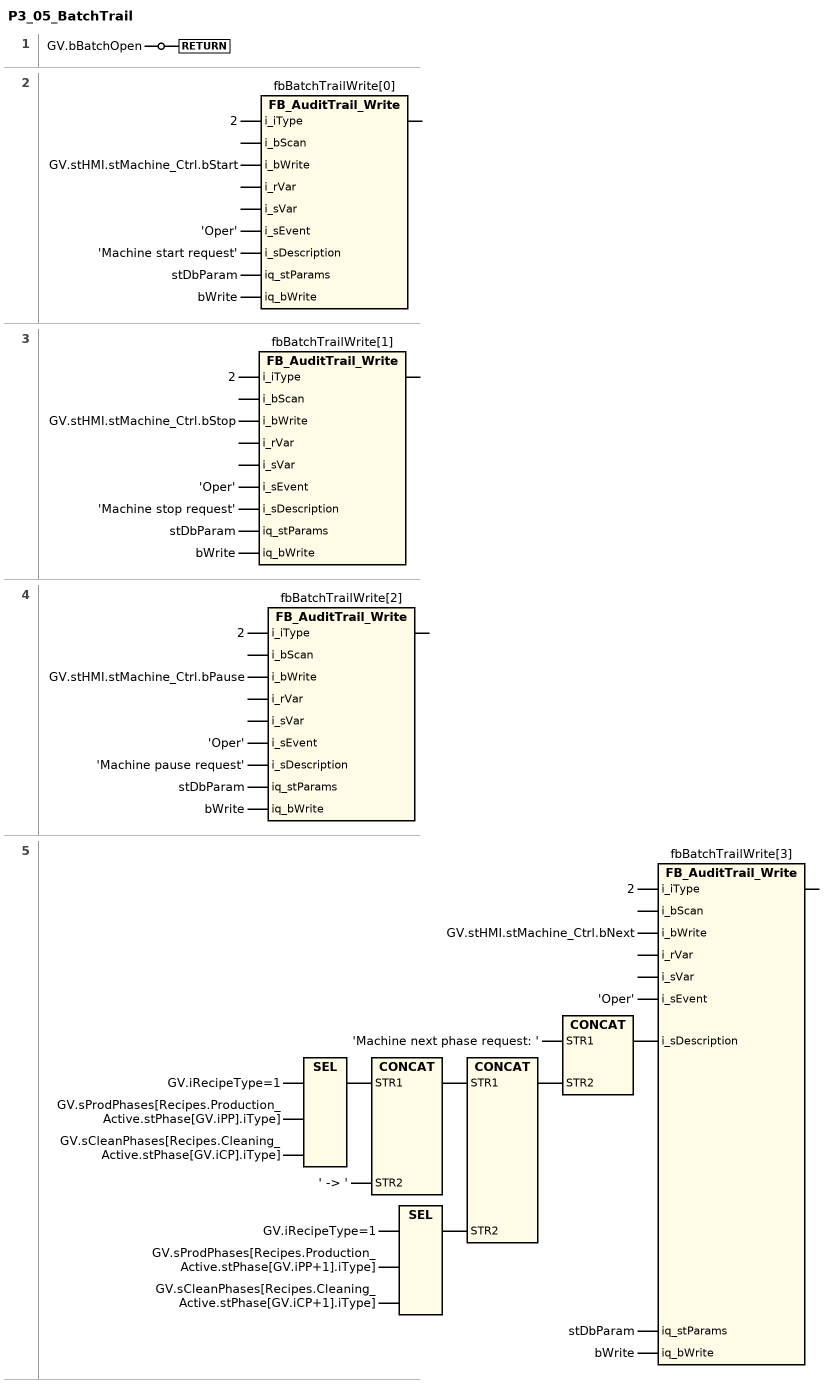
// NETWORK 1
IF NOT GV.bBatchOpen THEN RETURN; END_IF

// NETWORK 2
fbBatchTrailWrite[0](
    i_iType := 2,
    i_bWrite := GV.stHMI.stMachine_Ctrl.bStart,
    i_sEvent := 'Oper',
    i_sDescription := 'Machine start request',
    iq_stParams := stDbParam,
    iq_bWrite := bWrite); // FB_AuditTrail_Write

// NETWORK 3
fbBatchTrailWrite[1](
    i_iType := 2,
    i_bWrite := GV.stHMI.stMachine_Ctrl.bStop,
    i_sEvent := 'Oper',
    i_sDescription := 'Machine stop request',
    iq_stParams := stDbParam,
    iq_bWrite := bWrite); // FB_AuditTrail_Write

// NETWORK 4
fbBatchTrailWrite[2](
    i_iType := 2,
    i_bWrite := GV.stHMI.stMachine_Ctrl.bPause,
    i_sEvent := 'Oper',
    i_sDescription := 'Machine pause request',
    iq_stParams := stDbParam,
    iq_bWrite := bWrite); // FB_AuditTrail_Write

// NETWORK 5
fbBatchTrailWrite[3](
    i_iType := 2,
    i_bWrite := GV.stHMI.stMachine_Ctrl.bNext,
    i_sEvent := 'Oper',
    i_sDescription := CONCAT(STR1 := 'Machine next phase request: ', STR2 := CONCAT(STR1 := CONCAT(STR1 := SEL(GV.iRecipeType=1, GV.sProdPhases[Recipes.Production_Active.stPhase[GV.iPP].iType], GV.sCleanPhases[Recipes.Cleaning_Active.stPhase[GV.iCP].iType]), STR2 := ' -> '), STR2 := SEL(GV.iRecipeType=1, GV.sProdPhases[Recipes.Production_Active.stPhase[GV.iPP+1].iType], GV.sCleanPhases[Recipes.Cleaning_Active.stPhase[GV.iCP+1].iType]))),
    iq_stParams := stDbParam,
    iq_bWrite := bWrite); // FB_AuditTrail_Write

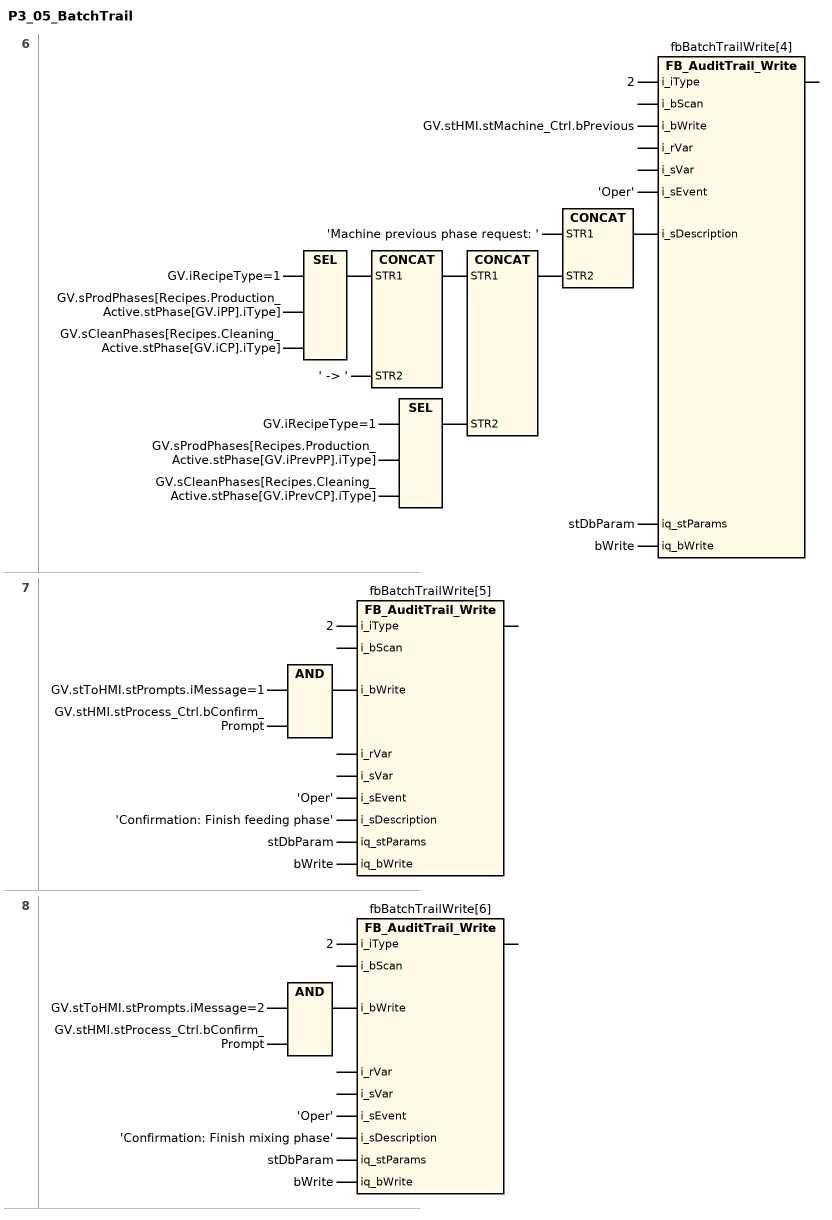
// NETWORK 6
fbBatchTrailWrite[4](
    i_iType := 2,
    i_bWrite := GV.stHMI.stMachine_Ctrl.bPrevious,
    i_sEvent := 'Oper',
    i_sDescription := CONCAT(STR1 := 'Machine previous phase request: ', STR2 := CONCAT(STR1 := CONCAT(STR1 := SEL(GV.iRecipeType=1, GV.sProdPhases[Recipes.Production_Active.stPhase[GV.iPP].iType], GV.sCleanPhases[Recipes.Cleaning_Active.stPhase[GV.iCP].iType]), STR2 := ' -> '), STR2 := SEL(GV.iRecipeType=1, GV.sProdPhases[Recipes.Production_Active.stPhase[GV.iPrevPP].iType], GV.sCleanPhases[Recipes.Cleaning_Active.stPhase[GV.iPrevCP].iType]))),
    iq_stParams := stDbParam,
    iq_bWrite := bWrite); // FB_AuditTrail_Write

// NETWORK 7
fbBatchTrailWrite[5](
    i_iType := 2,
    i_bWrite := (GV.stToHMI.stPrompts.iMessage=1) AND GV.stHMI.stProcess_Ctrl.bConfirm_Prompt,
    i_sEvent := 'Oper',
    i_sDescription := 'Confirmation: Finish feeding phase',
    iq_stParams := stDbParam,
    iq_bWrite := bWrite); // FB_AuditTrail_Write

// NETWORK 8
fbBatchTrailWrite[6](
    i_iType := 2,
    i_bWrite := (GV.stToHMI.stPrompts.iMessage=2) AND GV.stHMI.stProcess_Ctrl.bConfirm_Prompt,
    i_sEvent := 'Oper',
    i_sDescription := 'Confirmation: Finish mixing phase',
    iq_stParams := stDbParam,
    iq_bWrite := bWrite); // FB_AuditTrail_Write

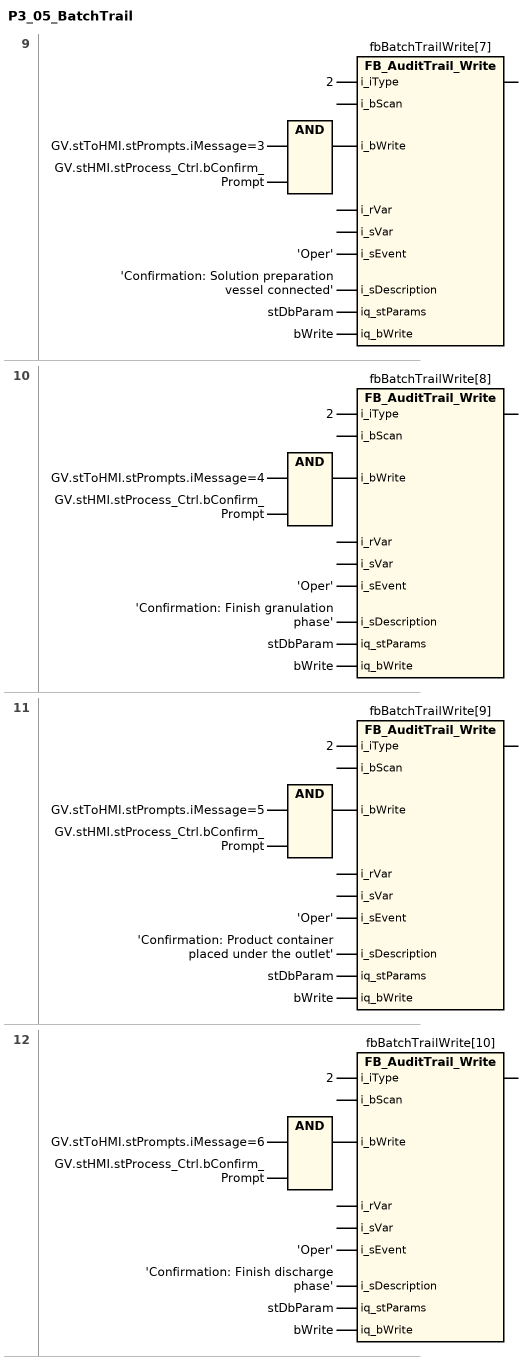
// NETWORK 9
fbBatchTrailWrite[7](
    i_iType := 2,
    i_bWrite := (GV.stToHMI.stPrompts.iMessage=3) AND GV.stHMI.stProcess_Ctrl.bConfirm_Prompt,
    i_sEvent := 'Oper',
    i_sDescription := 'Confirmation: Solution preparation vessel connected',
    iq_stParams := stDbParam,
    iq_bWrite := bWrite); // FB_AuditTrail_Write

// NETWORK 10
fbBatchTrailWrite[8](
    i_iType := 2,
    i_bWrite := (GV.stToHMI.stPrompts.iMessage=4) AND GV.stHMI.stProcess_Ctrl.bConfirm_Prompt,
    i_sEvent := 'Oper',
    i_sDescription := 'Confirmation: Finish granulation phase',
    iq_stParams := stDbParam,
    iq_bWrite := bWrite); // FB_AuditTrail_Write

// NETWORK 11
fbBatchTrailWrite[9](
    i_iType := 2,
    i_bWrite := (GV.stToHMI.stPrompts.iMessage=5) AND GV.stHMI.stProcess_Ctrl.bConfirm_Prompt,
    i_sEvent := 'Oper',
    i_sDescription := 'Confirmation: Product container placed under the outlet',
    iq_stParams := stDbParam,
    iq_bWrite := bWrite); // FB_AuditTrail_Write

// NETWORK 12
fbBatchTrailWrite[10](
    i_iType := 2,
    i_bWrite := (GV.stToHMI.stPrompts.iMessage=6) AND GV.stHMI.stProcess_Ctrl.bConfirm_Prompt,
    i_sEvent := 'Oper',
    i_sDescription := 'Confirmation: Finish discharge phase',
    iq_stParams := stDbParam,
    iq_bWrite := bWrite); // FB_AuditTrail_Write

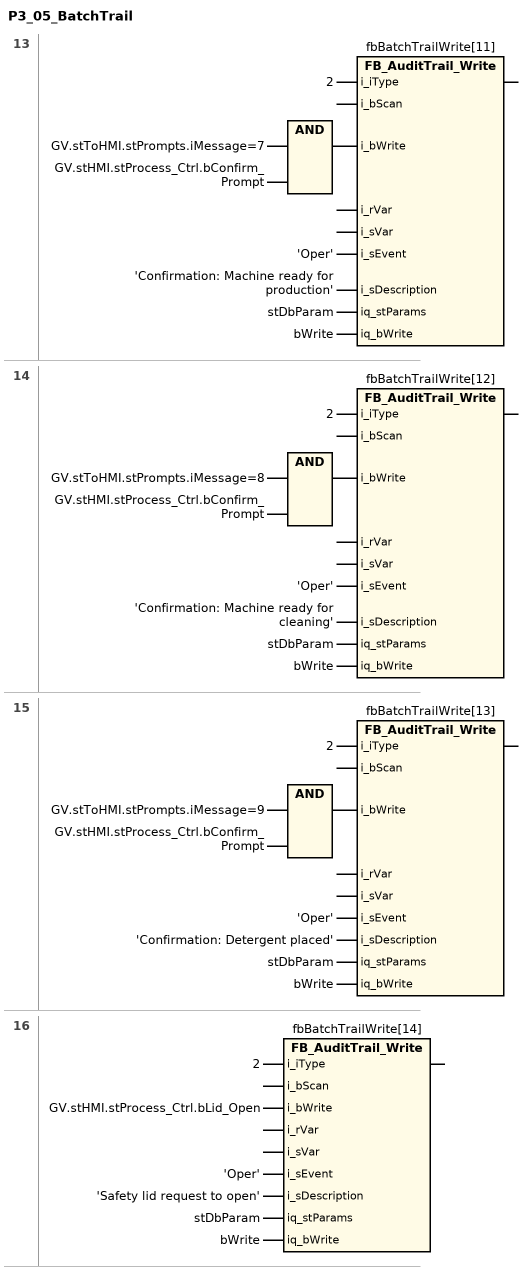
// NETWORK 13
fbBatchTrailWrite[11](
    i_iType := 2,
    i_bWrite := (GV.stToHMI.stPrompts.iMessage=7) AND GV.stHMI.stProcess_Ctrl.bConfirm_Prompt,
    i_sEvent := 'Oper',
    i_sDescription := 'Confirmation: Machine ready for production',
    iq_stParams := stDbParam,
    iq_bWrite := bWrite); // FB_AuditTrail_Write

// NETWORK 14
fbBatchTrailWrite[12](
    i_iType := 2,
    i_bWrite := (GV.stToHMI.stPrompts.iMessage=8) AND GV.stHMI.stProcess_Ctrl.bConfirm_Prompt,
    i_sEvent := 'Oper',
    i_sDescription := 'Confirmation: Machine ready for cleaning',
    iq_stParams := stDbParam,
    iq_bWrite := bWrite); // FB_AuditTrail_Write

// NETWORK 15
fbBatchTrailWrite[13](
    i_iType := 2,
    i_bWrite := (GV.stToHMI.stPrompts.iMessage=9) AND GV.stHMI.stProcess_Ctrl.bConfirm_Prompt,
    i_sEvent := 'Oper',
    i_sDescription := 'Confirmation: Detergent placed',
    iq_stParams := stDbParam,
    iq_bWrite := bWrite); // FB_AuditTrail_Write

// NETWORK 16
fbBatchTrailWrite[14](
    i_iType := 2,
    i_bWrite := GV.stHMI.stProcess_Ctrl.bLid_Open,
    i_sEvent := 'Oper',
    i_sDescription := 'Safety lid request to open',
    iq_stParams := stDbParam,
    iq_bWrite := bWrite); // FB_AuditTrail_Write

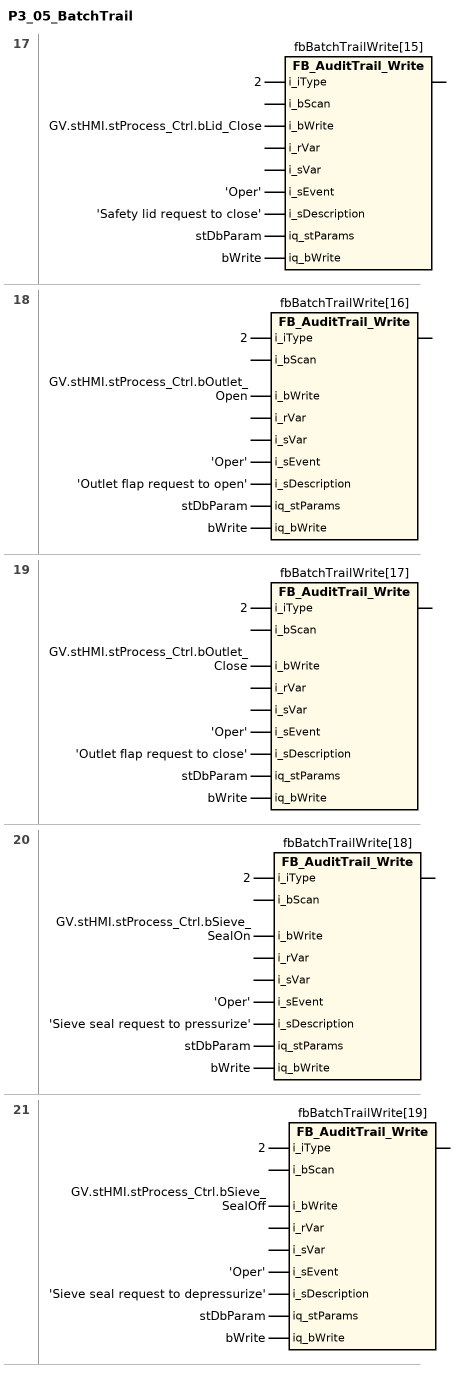
// NETWORK 17
fbBatchTrailWrite[15](
    i_iType := 2,
    i_bWrite := GV.stHMI.stProcess_Ctrl.bLid_Close,
    i_sEvent := 'Oper',
    i_sDescription := 'Safety lid request to close',
    iq_stParams := stDbParam,
    iq_bWrite := bWrite); // FB_AuditTrail_Write

// NETWORK 18
fbBatchTrailWrite[16](
    i_iType := 2,
    i_bWrite := GV.stHMI.stProcess_Ctrl.bOutlet_Open,
    i_sEvent := 'Oper',
    i_sDescription := 'Outlet flap request to open',
    iq_stParams := stDbParam,
    iq_bWrite := bWrite); // FB_AuditTrail_Write

// NETWORK 19
fbBatchTrailWrite[17](
    i_iType := 2,
    i_bWrite := GV.stHMI.stProcess_Ctrl.bOutlet_Close,
    i_sEvent := 'Oper',
    i_sDescription := 'Outlet flap request to close',
    iq_stParams := stDbParam,
    iq_bWrite := bWrite); // FB_AuditTrail_Write

// NETWORK 20
fbBatchTrailWrite[18](
    i_iType := 2,
    i_bWrite := GV.stHMI.stProcess_Ctrl.bSieve_SealOn,
    i_sEvent := 'Oper',
    i_sDescription := 'Sieve seal request to pressurize',
    iq_stParams := stDbParam,
    iq_bWrite := bWrite); // FB_AuditTrail_Write

// NETWORK 21
fbBatchTrailWrite[19](
    i_iType := 2,
    i_bWrite := GV.stHMI.stProcess_Ctrl.bSieve_SealOff,
    i_sEvent := 'Oper',
    i_sDescription := 'Sieve seal request to depressurize',
    iq_stParams := stDbParam,
    iq_bWrite := bWrite); // FB_AuditTrail_Write

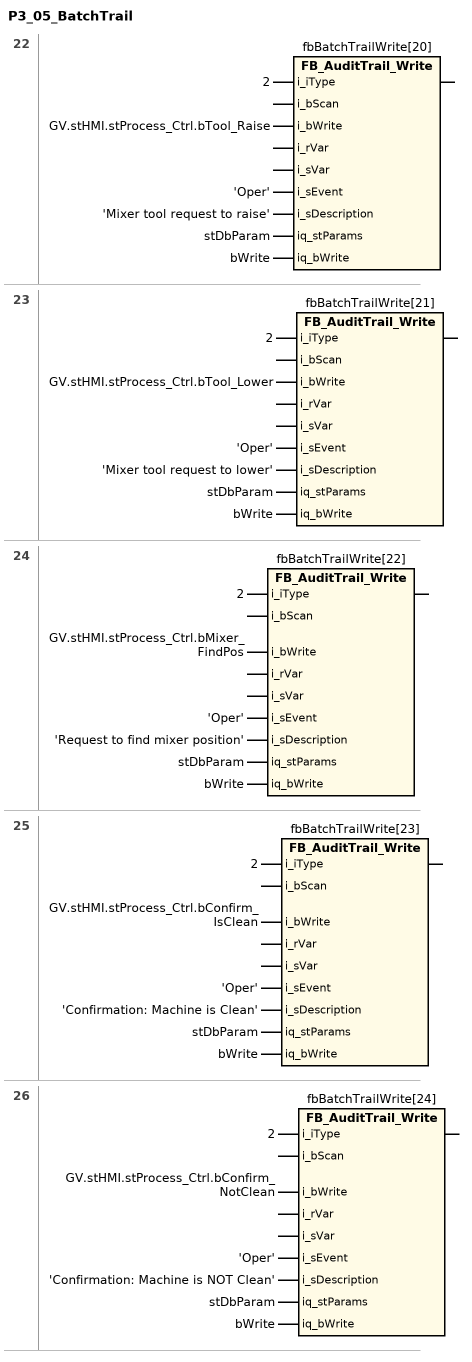
// NETWORK 22
fbBatchTrailWrite[20](
    i_iType := 2,
    i_bWrite := GV.stHMI.stProcess_Ctrl.bTool_Raise,
    i_sEvent := 'Oper',
    i_sDescription := 'Mixer tool request to raise',
    iq_stParams := stDbParam,
    iq_bWrite := bWrite); // FB_AuditTrail_Write

// NETWORK 23
fbBatchTrailWrite[21](
    i_iType := 2,
    i_bWrite := GV.stHMI.stProcess_Ctrl.bTool_Lower,
    i_sEvent := 'Oper',
    i_sDescription := 'Mixer tool request to lower',
    iq_stParams := stDbParam,
    iq_bWrite := bWrite); // FB_AuditTrail_Write

// NETWORK 24
fbBatchTrailWrite[22](
    i_iType := 2,
    i_bWrite := GV.stHMI.stProcess_Ctrl.bMixer_FindPos,
    i_sEvent := 'Oper',
    i_sDescription := 'Request to find mixer position',
    iq_stParams := stDbParam,
    iq_bWrite := bWrite); // FB_AuditTrail_Write

// NETWORK 25
fbBatchTrailWrite[23](
    i_iType := 2,
    i_bWrite := GV.stHMI.stProcess_Ctrl.bConfirm_IsClean,
    i_sEvent := 'Oper',
    i_sDescription := 'Confirmation: Machine is Clean',
    iq_stParams := stDbParam,
    iq_bWrite := bWrite); // FB_AuditTrail_Write

// NETWORK 26
fbBatchTrailWrite[24](
    i_iType := 2,
    i_bWrite := GV.stHMI.stProcess_Ctrl.bConfirm_NotClean,
    i_sEvent := 'Oper',
    i_sDescription := 'Confirmation: Machine is NOT Clean',
    iq_stParams := stDbParam,
    iq_bWrite := bWrite); // FB_AuditTrail_Write

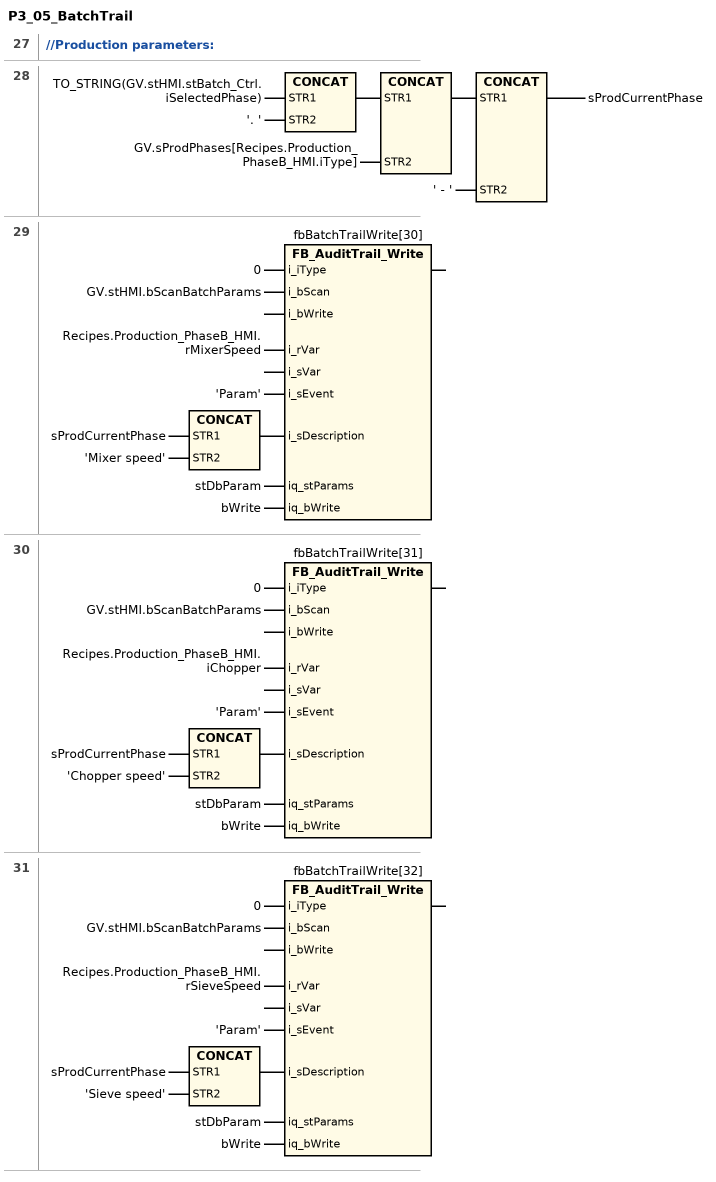
// NETWORK 27
// label: //Production parameters

// NETWORK 28
sProdCurrentPhase := CONCAT(STR1 := CONCAT(STR1 := CONCAT(STR1 := TO_STRING(GV.stHMI.stBatch_Ctrl.iSelectedPhase), STR2 := '. '), STR2 := GV.sProdPhases[Recipes.Production_PhaseB_HMI.iType]), STR2 := ' - ');

// NETWORK 29
fbBatchTrailWrite[30](
    i_iType := 0,
    i_bScan := GV.stHMI.bScanBatchParams,
    i_rVar := Recipes.Production_PhaseB_HMI.rMixerSpeed,
    i_sEvent := 'Param',
    i_sDescription := CONCAT(STR1 := sProdCurrentPhase, STR2 := 'Mixer speed'),
    iq_stParams := stDbParam,
    iq_bWrite := bWrite); // FB_AuditTrail_Write

// NETWORK 30
fbBatchTrailWrite[31](
    i_iType := 0,
    i_bScan := GV.stHMI.bScanBatchParams,
    i_rVar := Recipes.Production_PhaseB_HMI.iChopper,
    i_sEvent := 'Param',
    i_sDescription := CONCAT(STR1 := sProdCurrentPhase, STR2 := 'Chopper speed'),
    iq_stParams := stDbParam,
    iq_bWrite := bWrite); // FB_AuditTrail_Write

// NETWORK 31
fbBatchTrailWrite[32](
    i_iType := 0,
    i_bScan := GV.stHMI.bScanBatchParams,
    i_rVar := Recipes.Production_PhaseB_HMI.rSieveSpeed,
    i_sEvent := 'Param',
    i_sDescription := CONCAT(STR1 := sProdCurrentPhase, STR2 := 'Sieve speed'),
    iq_stParams := stDbParam,
    iq_bWrite := bWrite); // FB_AuditTrail_Write

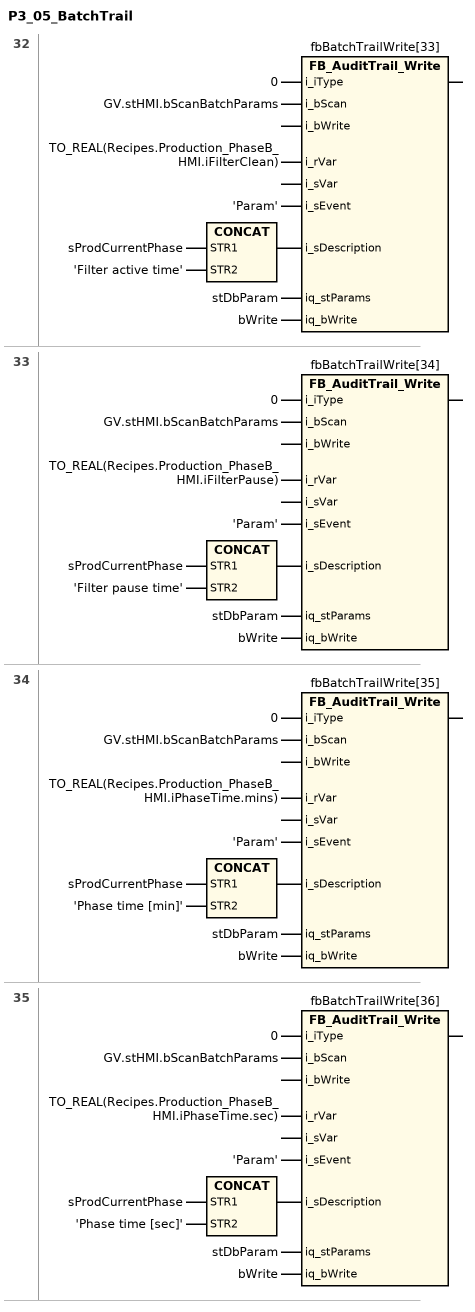
// NETWORK 32
fbBatchTrailWrite[33](
    i_iType := 0,
    i_bScan := GV.stHMI.bScanBatchParams,
    i_rVar := TO_REAL(Recipes.Production_PhaseB_HMI.iFilterClean),
    i_sEvent := 'Param',
    i_sDescription := CONCAT(STR1 := sProdCurrentPhase, STR2 := 'Filter active time'),
    iq_stParams := stDbParam,
    iq_bWrite := bWrite); // FB_AuditTrail_Write

// NETWORK 33
fbBatchTrailWrite[34](
    i_iType := 0,
    i_bScan := GV.stHMI.bScanBatchParams,
    i_rVar := TO_REAL(Recipes.Production_PhaseB_HMI.iFilterPause),
    i_sEvent := 'Param',
    i_sDescription := CONCAT(STR1 := sProdCurrentPhase, STR2 := 'Filter pause time'),
    iq_stParams := stDbParam,
    iq_bWrite := bWrite); // FB_AuditTrail_Write

// NETWORK 34
fbBatchTrailWrite[35](
    i_iType := 0,
    i_bScan := GV.stHMI.bScanBatchParams,
    i_rVar := TO_REAL(Recipes.Production_PhaseB_HMI.iPhaseTime.mins),
    i_sEvent := 'Param',
    i_sDescription := CONCAT(STR1 := sProdCurrentPhase, STR2 := 'Phase time [min]'),
    iq_stParams := stDbParam,
    iq_bWrite := bWrite); // FB_AuditTrail_Write

// NETWORK 35
fbBatchTrailWrite[36](
    i_iType := 0,
    i_bScan := GV.stHMI.bScanBatchParams,
    i_rVar := TO_REAL(Recipes.Production_PhaseB_HMI.iPhaseTime.sec),
    i_sEvent := 'Param',
    i_sDescription := CONCAT(STR1 := sProdCurrentPhase, STR2 := 'Phase time [sec]'),
    iq_stParams := stDbParam,
    iq_bWrite := bWrite); // FB_AuditTrail_Write

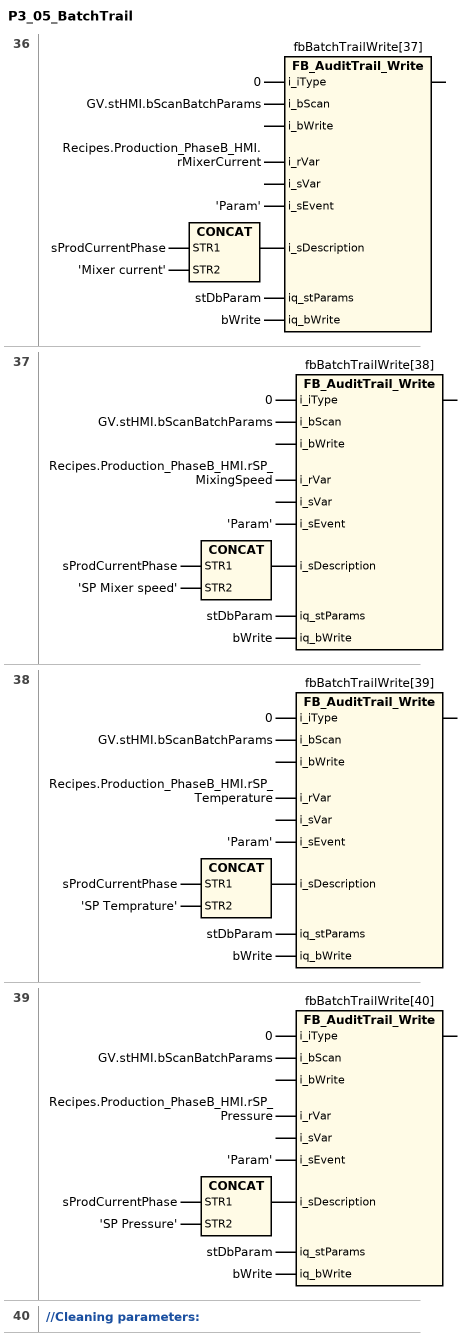
// NETWORK 36
fbBatchTrailWrite[37](
    i_iType := 0,
    i_bScan := GV.stHMI.bScanBatchParams,
    i_rVar := Recipes.Production_PhaseB_HMI.rMixerCurrent,
    i_sEvent := 'Param',
    i_sDescription := CONCAT(STR1 := sProdCurrentPhase, STR2 := 'Mixer current'),
    iq_stParams := stDbParam,
    iq_bWrite := bWrite); // FB_AuditTrail_Write

// NETWORK 37
fbBatchTrailWrite[38](
    i_iType := 0,
    i_bScan := GV.stHMI.bScanBatchParams,
    i_rVar := Recipes.Production_PhaseB_HMI.rSP_MixingSpeed,
    i_sEvent := 'Param',
    i_sDescription := CONCAT(STR1 := sProdCurrentPhase, STR2 := 'SP Mixer speed'),
    iq_stParams := stDbParam,
    iq_bWrite := bWrite); // FB_AuditTrail_Write

// NETWORK 38
fbBatchTrailWrite[39](
    i_iType := 0,
    i_bScan := GV.stHMI.bScanBatchParams,
    i_rVar := Recipes.Production_PhaseB_HMI.rSP_Temperature,
    i_sEvent := 'Param',
    i_sDescription := CONCAT(STR1 := sProdCurrentPhase, STR2 := 'SP Temprature'),
    iq_stParams := stDbParam,
    iq_bWrite := bWrite); // FB_AuditTrail_Write

// NETWORK 39
fbBatchTrailWrite[40](
    i_iType := 0,
    i_bScan := GV.stHMI.bScanBatchParams,
    i_rVar := Recipes.Production_PhaseB_HMI.rSP_Pressure,
    i_sEvent := 'Param',
    i_sDescription := CONCAT(STR1 := sProdCurrentPhase, STR2 := 'SP Pressure'),
    iq_stParams := stDbParam,
    iq_bWrite := bWrite); // FB_AuditTrail_Write

// NETWORK 40
// label: //Cleaning parameters

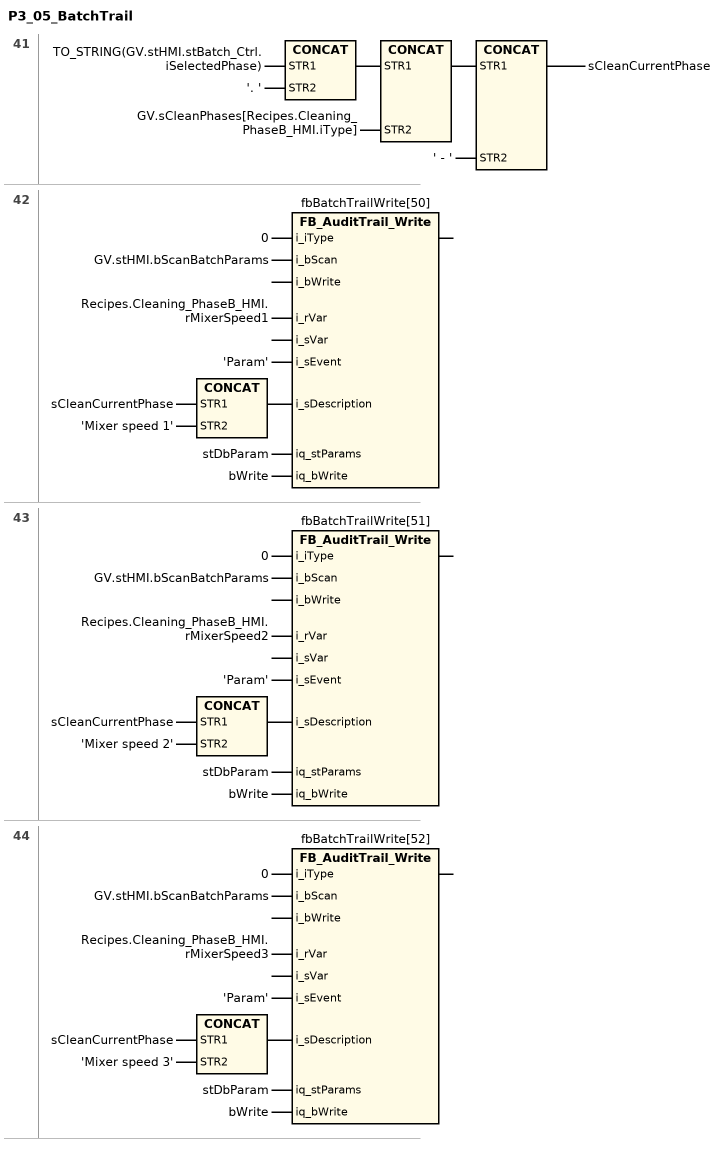
// NETWORK 41
sCleanCurrentPhase := CONCAT(STR1 := CONCAT(STR1 := CONCAT(STR1 := TO_STRING(GV.stHMI.stBatch_Ctrl.iSelectedPhase), STR2 := '. '), STR2 := GV.sCleanPhases[Recipes.Cleaning_PhaseB_HMI.iType]), STR2 := ' - ');

// NETWORK 42
fbBatchTrailWrite[50](
    i_iType := 0,
    i_bScan := GV.stHMI.bScanBatchParams,
    i_rVar := Recipes.Cleaning_PhaseB_HMI.rMixerSpeed1,
    i_sEvent := 'Param',
    i_sDescription := CONCAT(STR1 := sCleanCurrentPhase, STR2 := 'Mixer speed 1'),
    iq_stParams := stDbParam,
    iq_bWrite := bWrite); // FB_AuditTrail_Write

// NETWORK 43
fbBatchTrailWrite[51](
    i_iType := 0,
    i_bScan := GV.stHMI.bScanBatchParams,
    i_rVar := Recipes.Cleaning_PhaseB_HMI.rMixerSpeed2,
    i_sEvent := 'Param',
    i_sDescription := CONCAT(STR1 := sCleanCurrentPhase, STR2 := 'Mixer speed 2'),
    iq_stParams := stDbParam,
    iq_bWrite := bWrite); // FB_AuditTrail_Write

// NETWORK 44
fbBatchTrailWrite[52](
    i_iType := 0,
    i_bScan := GV.stHMI.bScanBatchParams,
    i_rVar := Recipes.Cleaning_PhaseB_HMI.rMixerSpeed3,
    i_sEvent := 'Param',
    i_sDescription := CONCAT(STR1 := sCleanCurrentPhase, STR2 := 'Mixer speed 3'),
    iq_stParams := stDbParam,
    iq_bWrite := bWrite); // FB_AuditTrail_Write

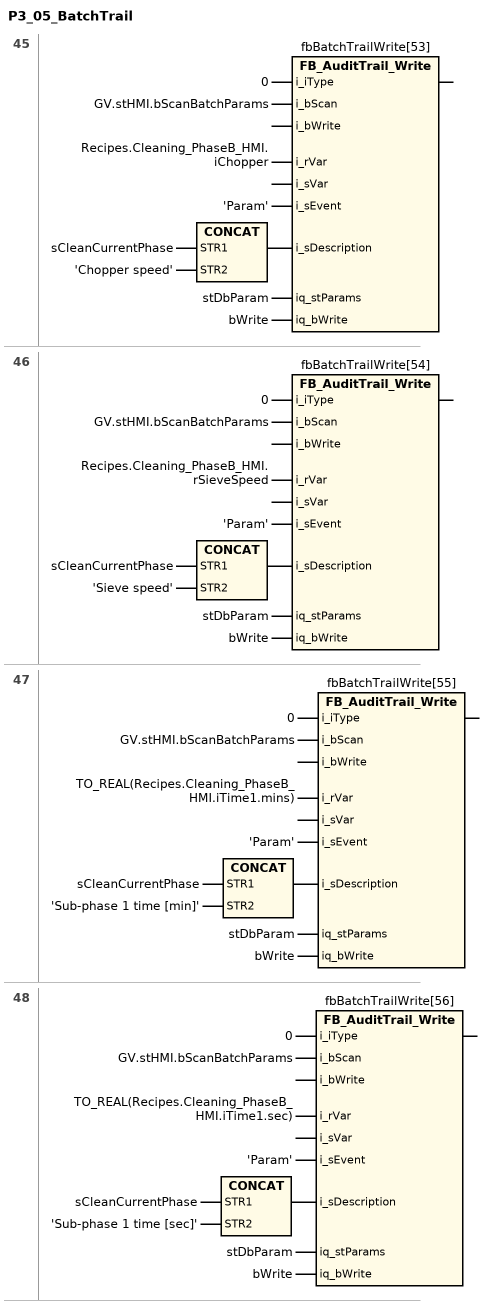
// NETWORK 45
fbBatchTrailWrite[53](
    i_iType := 0,
    i_bScan := GV.stHMI.bScanBatchParams,
    i_rVar := Recipes.Cleaning_PhaseB_HMI.iChopper,
    i_sEvent := 'Param',
    i_sDescription := CONCAT(STR1 := sCleanCurrentPhase, STR2 := 'Chopper speed'),
    iq_stParams := stDbParam,
    iq_bWrite := bWrite); // FB_AuditTrail_Write

// NETWORK 46
fbBatchTrailWrite[54](
    i_iType := 0,
    i_bScan := GV.stHMI.bScanBatchParams,
    i_rVar := Recipes.Cleaning_PhaseB_HMI.rSieveSpeed,
    i_sEvent := 'Param',
    i_sDescription := CONCAT(STR1 := sCleanCurrentPhase, STR2 := 'Sieve speed'),
    iq_stParams := stDbParam,
    iq_bWrite := bWrite); // FB_AuditTrail_Write

// NETWORK 47
fbBatchTrailWrite[55](
    i_iType := 0,
    i_bScan := GV.stHMI.bScanBatchParams,
    i_rVar := TO_REAL(Recipes.Cleaning_PhaseB_HMI.iTime1.mins),
    i_sEvent := 'Param',
    i_sDescription := CONCAT(STR1 := sCleanCurrentPhase, STR2 := 'Sub-phase 1 time [min]'),
    iq_stParams := stDbParam,
    iq_bWrite := bWrite); // FB_AuditTrail_Write

// NETWORK 48
fbBatchTrailWrite[56](
    i_iType := 0,
    i_bScan := GV.stHMI.bScanBatchParams,
    i_rVar := TO_REAL(Recipes.Cleaning_PhaseB_HMI.iTime1.sec),
    i_sEvent := 'Param',
    i_sDescription := CONCAT(STR1 := sCleanCurrentPhase, STR2 := 'Sub-phase 1 time [sec]'),
    iq_stParams := stDbParam,
    iq_bWrite := bWrite); // FB_AuditTrail_Write

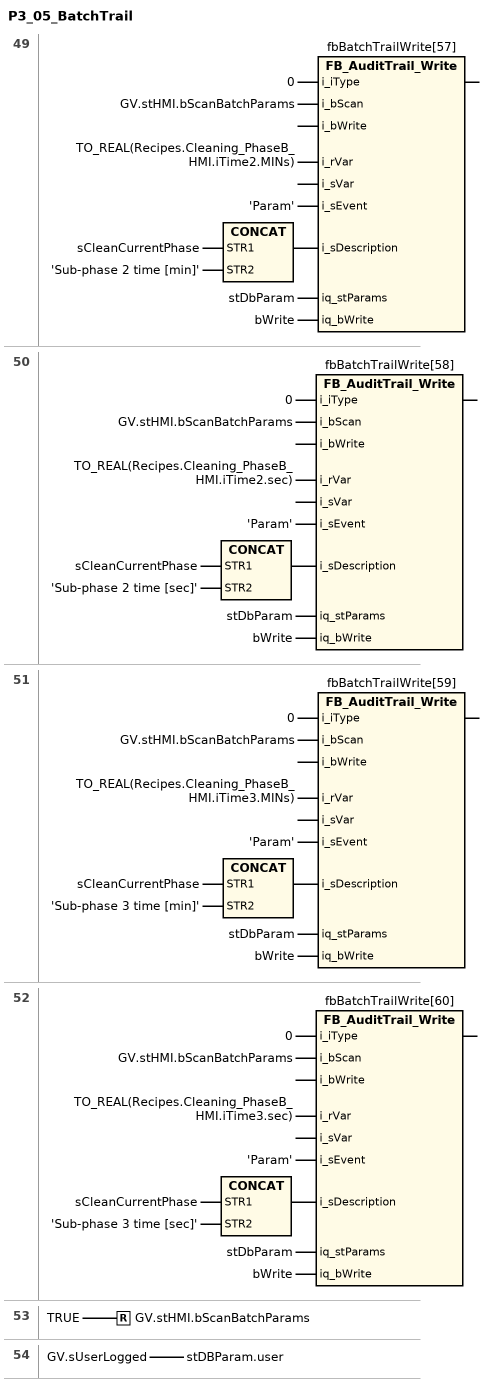
// NETWORK 49
fbBatchTrailWrite[57](
    i_iType := 0,
    i_bScan := GV.stHMI.bScanBatchParams,
    i_rVar := TO_REAL(Recipes.Cleaning_PhaseB_HMI.iTime2.MINs),
    i_sEvent := 'Param',
    i_sDescription := CONCAT(STR1 := sCleanCurrentPhase, STR2 := 'Sub-phase 2 time [min]'),
    iq_stParams := stDbParam,
    iq_bWrite := bWrite); // FB_AuditTrail_Write

// NETWORK 50
fbBatchTrailWrite[58](
    i_iType := 0,
    i_bScan := GV.stHMI.bScanBatchParams,
    i_rVar := TO_REAL(Recipes.Cleaning_PhaseB_HMI.iTime2.sec),
    i_sEvent := 'Param',
    i_sDescription := CONCAT(STR1 := sCleanCurrentPhase, STR2 := 'Sub-phase 2 time [sec]'),
    iq_stParams := stDbParam,
    iq_bWrite := bWrite); // FB_AuditTrail_Write

// NETWORK 51
fbBatchTrailWrite[59](
    i_iType := 0,
    i_bScan := GV.stHMI.bScanBatchParams,
    i_rVar := TO_REAL(Recipes.Cleaning_PhaseB_HMI.iTime3.MINs),
    i_sEvent := 'Param',
    i_sDescription := CONCAT(STR1 := sCleanCurrentPhase, STR2 := 'Sub-phase 3 time [min]'),
    iq_stParams := stDbParam,
    iq_bWrite := bWrite); // FB_AuditTrail_Write

// NETWORK 52
fbBatchTrailWrite[60](
    i_iType := 0,
    i_bScan := GV.stHMI.bScanBatchParams,
    i_rVar := TO_REAL(Recipes.Cleaning_PhaseB_HMI.iTime3.sec),
    i_sEvent := 'Param',
    i_sDescription := CONCAT(STR1 := sCleanCurrentPhase, STR2 := 'Sub-phase 3 time [sec]'),
    iq_stParams := stDbParam,
    iq_bWrite := bWrite); // FB_AuditTrail_Write

// NETWORK 53
GV.stHMI.bScanBatchParams R= TRUE;

// NETWORK 54
stDBParam.user := GV.sUserLogged;

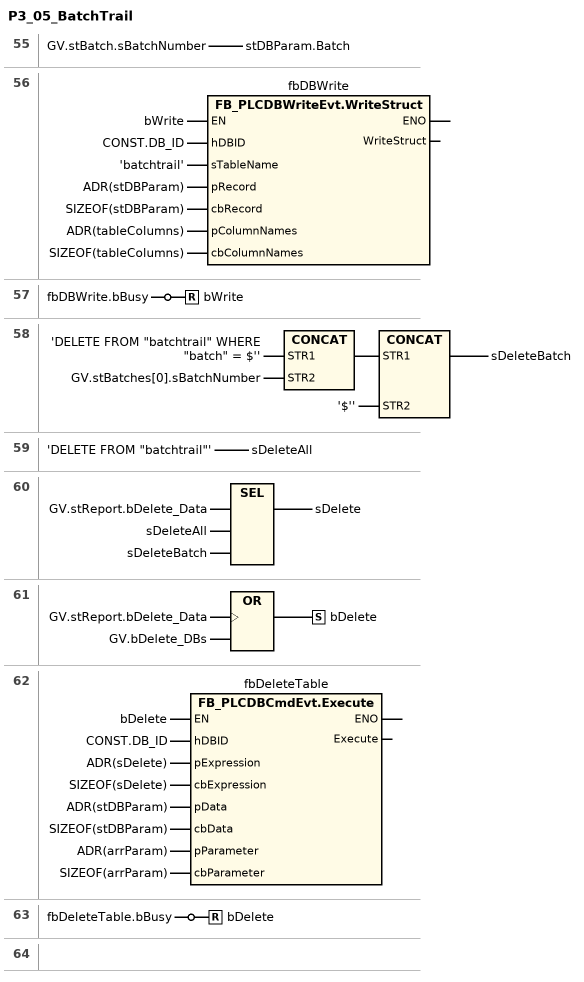
// NETWORK 55
stDBParam.Batch := GV.stBatch.sBatchNumber;

// NETWORK 56
IF bWrite THEN
    fbDBWrite.WriteStruct(
        hDBID := CONST.DB_ID,
        sTableName := 'batchtrail',
        pRecord := ADR(stDBParam),
        cbRecord := SIZEOF(stDBParam),
        pColumnNames := ADR(tableColumns),
        cbColumnNames := SIZEOF(tableColumns));
END_IF

// NETWORK 57
bWrite R= NOT fbDBWrite.bBusy;

// NETWORK 58
sDeleteBatch := CONCAT(STR1 := CONCAT(STR1 := 'DELETE FROM "batchtrail" WHERE "batch" = $'', STR2 := GV.stBatches[0].sBatchNumber), STR2 := '$'');

// NETWORK 59
sDeleteAll := 'DELETE FROM "batchtrail"';

// NETWORK 60
sDelete := SEL(GV.stReport.bDelete_Data, sDeleteAll, sDeleteBatch);

// NETWORK 61
_rt1(CLK := GV.stReport.bDelete_Data);
bDelete S= _rt1.Q OR GV.bDelete_DBs;

// NETWORK 62
IF bDelete THEN
    fbDeleteTable.Execute(
        hDBID := CONST.DB_ID,
        pExpression := ADR(sDelete),
        cbExpression := SIZEOF(sDelete),
        pData := ADR(stDBParam),
        cbData := SIZEOF(stDBParam),
        pParameter := ADR(arrParam),
        cbParameter := SIZEOF(arrParam));
END_IF

// NETWORK 63
bDelete R= NOT fbDeleteTable.bBusy;

// NETWORK 64

END_PROGRAM

// ---- FBs/FB_AuditTrail_Write.TcPOU
FUNCTION_BLOCK FB_AuditTrail_Write
VAR_INPUT
	i_iType			:INT; //0-REAL,1-STRING,2-BOOL
	i_bScan			:BOOL;
	i_bWrite		:BOOL;
	i_rVar			:REAL;
	i_sVar			:STRING;
	i_sEvent		:STRING;
	i_sDescription	:STRING;
END_VAR
VAR
	iVarOld			:REAL;
	sVarOld			:STRING;
	bVarOld			:BOOL;
	bScan			:BOOL;
	Scan_TON		:TON;
END_VAR
VAR_IN_OUT
	iq_stParams		:ST_BatchTrail;
	iq_bWrite		:BOOL;
END_VAR

IF i_iType = 0 THEN
	ACT_REAL();
ELSIF i_iType = 1 THEN
	ACT_STRING();
ELSIF i_iType = 2 THEN
	ACT_BOOL();
END_IF

ACTION ACT_BOOL:
IF i_bWrite THEN
	iq_stParams.Event:=i_sEvent;
	iq_stParams.Description := i_sDescription;
	iq_stParams.Oldvalue:='/';
	iq_stParams.Newvalue:='/';
	iq_bWrite:=TRUE;
END_IF
END_ACTION

ACTION ACT_REAL:
IF i_bScan THEN
	bScan:=TRUE;
END_IF
Scan_TON(IN:=bScan,PT:=T#3S);
IF Scan_TON.Q THEN
	iVarOld:=i_rVar;
	bScan:=FALSE;
END_IF
IF NOT bScan AND iVarOld <> i_rVar THEN
	iq_stParams.Event:=i_sEvent;
	iq_stParams.Description := i_sDescription;
	iq_stParams.Oldvalue:=REAL_TO_STRING(iVarOld);
	iq_stParams.Newvalue:=REAL_TO_STRING(i_rVar);
	iVarOld:=i_rVar;
	iq_bWrite:=TRUE;
END_IF
END_ACTION

ACTION ACT_STRING:
IF i_bScan THEN
	bScan:=TRUE;
END_IF
Scan_TON(IN:=bScan,PT:=T#3S);
IF Scan_TON.Q THEN
	sVarOld:=i_sVar;
	bScan:=FALSE;
END_IF
IF i_bWrite AND NOT bScan AND sVarOld <> i_sVar THEN
	iq_stParams.Event:=i_sEvent;
	iq_stParams.Description := i_sDescription;
	iq_stParams.Oldvalue:=sVarOld;
	iq_stParams.Newvalue:=i_sVar;
	sVarOld:=i_sVar;
	iq_bWrite:=TRUE;
END_IF
END_ACTION

END_FUNCTION_BLOCK

// ---- POUs/3. Report/P3_06_SP_CreateReport.TcPOU
PROGRAM P3_06_SP_CreateReport
VAR
	iStep					:INT;
	iError					:INT;
	tonResetError			:TON;
	trigStart				:R_TRIG;
	tonDelayStart			:TON;
	tonDelayDelete			:TON;
	
	fbReport				:FB_PythonScript;
END_VAR

ACT_CMDs();
trigStart(CLK:=GV.bSP_BatchClose);
IF tonResetError.Q THEN
	iError:=0;
END_IF

tonDelayStart(IN:=(iStep=10),PT:=T#1S);
tonDelayDelete(IN:=(iStep=999),PT:=T#1S);
CASE iStep OF
	
	0:
		IF trigStart.Q AND GV.stSP_Batch.sBatchName <> GV.sEmptyString AND NOT MAIn.bFirstCycle THEN
			iError:=0;
			iStep:=10;
		END_IF
		
	10:
		IF tonDelayStart.Q THEN
			iStep:=100;
		END_IF
		
	100:
		GV.stReport.bCreate_SPReport:=TRUE;
		IF fbReport.q_bBusy THEN
			iStep:=110;
		END_IF
	110:
		IF NOT fbReport.q_bBusy AND fbReport.q_bDone THEN
			iStep:=999;
		ELSIF fbReport.q_bError THEN
			iError:=iStep;
			iStep:=999;
		END_IF
	999:
		GV.stReport.bDelete_SPData:=TRUE;
		IF tonDelayDelete.Q THEN
			GV.stReport.bDelete_SPData:=FALSE;
			iStep:=0;
		END_IF
END_CASE

ACTION ACT_CMDs:
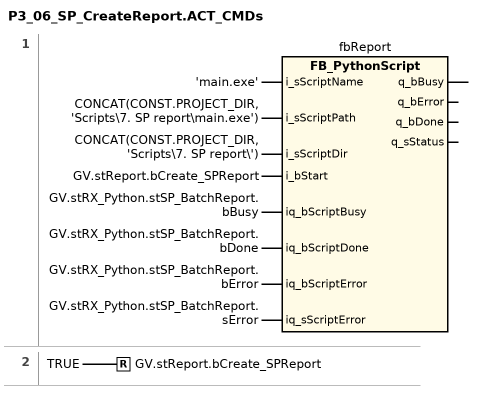
// NETWORK 1
fbReport(
    i_sScriptName := 'main.exe',
    i_sScriptPath := CONCAT(CONST.PROJECT_DIR,'Scripts\7. SP report\main.exe'),
    i_sScriptDir := CONCAT(CONST.PROJECT_DIR,'Scripts\7. SP report\'),
    i_bStart := GV.stReport.bCreate_SPReport,
    iq_bScriptBusy := GV.stRX_Python.stSP_BatchReport.bBusy,
    iq_bScriptDone := GV.stRX_Python.stSP_BatchReport.bDone,
    iq_bScriptError := GV.stRX_Python.stSP_BatchReport.bError,
    iq_sScriptError := GV.stRX_Python.stSP_BatchReport.sError); // FB_PythonScript

// NETWORK 2
GV.stReport.bCreate_SPReport R= TRUE;
END_ACTION

END_PROGRAM

// ---- POUs/3. Report/P3_07_SendReport.TcPOU
PROGRAM P3_07_SendReport
VAR
	fbSend				:FB_PythonScript;
	
	iError				:INT;
	tonResetError		:TON;
	
	iStep				:INT;
END_VAR

VAR PERSISTENT
	
END_VAR

tonResetError(IN:=(iError<>0),PT:=T#3S);
IF tonResetError.Q THEN
	iError:=0;
END_IF
CASE iStep OF
	
	0:
		IF GV.stReport.bStartSend_Sequence THEN
			GV.stReport.bStartSend_Sequence:=FALSE;
			iError:=0;
			iStep:=10;
		END_IF
	
	10:
		GV.stReport.bSend_Report:=TRUE;
		IF fbSend.q_bBusy THEN
			iStep:=15;
		END_IF
	
	15:
		IF NOT fbSend.q_bBusy AND fbSend.q_bDone THEN
			iStep:=999;
		ELSIF fbSend.q_bError THEN
			iError:=iStep;
			iStep:=999;
		END_IF
	
	999:
		iStep:=0;
END_CASE
ACT_CMDs();

ACTION ACT_CMDs:
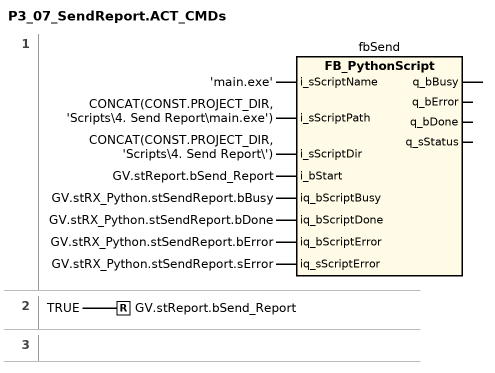
// NETWORK 1
fbSend(
    i_sScriptName := 'main.exe',
    i_sScriptPath := CONCAT(CONST.PROJECT_DIR,'Scripts\4. Send Report\main.exe'),
    i_sScriptDir := CONCAT(CONST.PROJECT_DIR,'Scripts\4. Send Report\'),
    i_bStart := GV.stReport.bSend_Report,
    iq_bScriptBusy := GV.stRX_Python.stSendReport.bBusy,
    iq_bScriptDone := GV.stRX_Python.stSendReport.bDone,
    iq_bScriptError := GV.stRX_Python.stSendReport.bError,
    iq_sScriptError := GV.stRX_Python.stSendReport.sError); // FB_PythonScript

// NETWORK 2
GV.stReport.bSend_Report R= TRUE;

// NETWORK 3
END_ACTION

END_PROGRAM

// ---- POUs/3. Report/P3_08_OpenReport.TcPOU
PROGRAM P3_08_OpenReport
VAR
	sDateTime			:STRING;
	sYear				:STRING;
	sMonth				:STRING;
	sDay				:STRING;
	sHour				:STRING;
	sMinute				:STRING;
	sReportSuffix		:STRING;
END_VAR

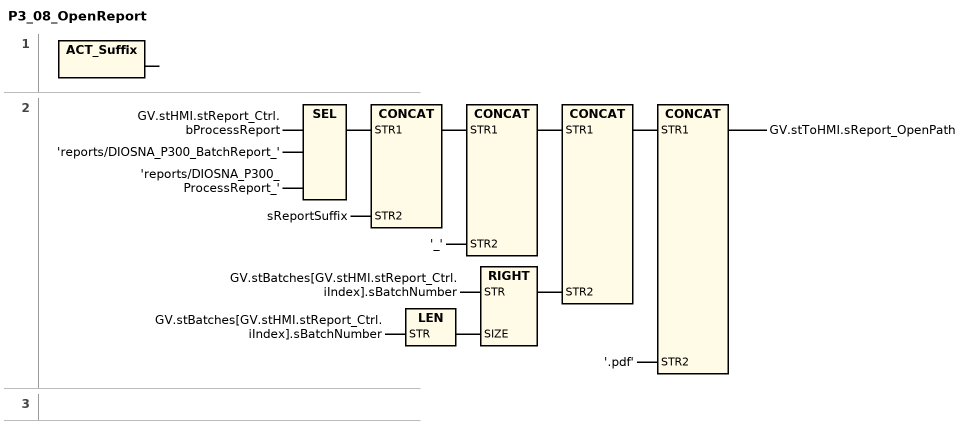
// NETWORK 1
ACT_Suffix();

// NETWORK 2
GV.stToHMI.sReport_OpenPath := CONCAT(STR1 := CONCAT(STR1 := CONCAT(STR1 := CONCAT(STR1 := SEL(GV.stHMI.stReport_Ctrl.bProcessReport, 'reports/DIOSNA_P300_BatchReport_', 'reports/DIOSNA_P300_ProcessReport_'), STR2 := sReportSuffix), STR2 := '_'), STR2 := RIGHT(STR := GV.stBatches[GV.stHMI.stReport_Ctrl.iIndex].sBatchNumber, SIZE := LEN(STR := GV.stBatches[GV.stHMI.stReport_Ctrl.iIndex].sBatchNumber))), STR2 := '.pdf');

// NETWORK 3

ACTION ACT_Suffix:
sDateTime:=GV.stBatches[GV.stHMI.stReport_Ctrl.iIndex].sFinished;
sYear:=RIGHT(LEFT(sDateTime,10),2);
sMonth:=RIGHT(LEFT(sDateTime,5),2);
sDay:=LEFT(sDateTime,2);

sHour:=LEFT(RIGHT(sDateTime,8),2);
sMinute:=LEFT(RIGHT(sDateTime,5),2);

sReportSuffix:=CONCAT(sYear,sMonth);
sReportSuffix:=CONCAT(sReportSuffix,sDay);
sReportSuffix:=CONCAT(sReportSuffix,sHour);
sReportSuffix:=CONCAT(sReportSuffix,sMinute);
END_ACTION

END_PROGRAM

// ---- POUs/5. HMI/P5_00_MAIN.TcPOU
PROGRAM P5_00_MAIN
VAR

END_VAR

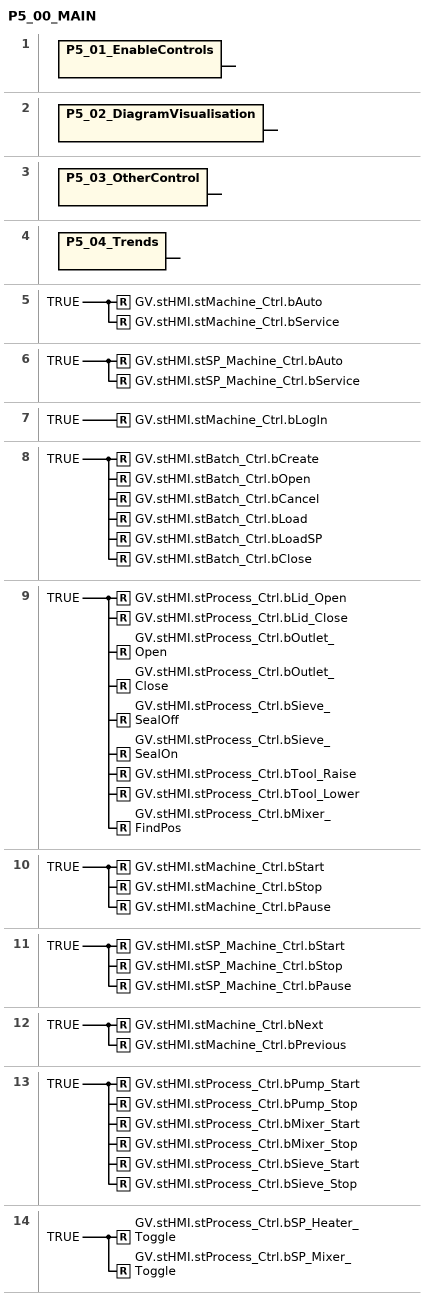
// NETWORK 1
P5_01_EnableControls();

// NETWORK 2
P5_02_DiagramVisualisation();

// NETWORK 3
P5_03_OtherControl();

// NETWORK 4
P5_04_Trends();

// NETWORK 5
GV.stHMI.stMachine_Ctrl.bAuto R= TRUE;
GV.stHMI.stMachine_Ctrl.bService R= TRUE;

// NETWORK 6
GV.stHMI.stSP_Machine_Ctrl.bAuto R= TRUE;
GV.stHMI.stSP_Machine_Ctrl.bService R= TRUE;

// NETWORK 7
GV.stHMI.stMachine_Ctrl.bLogIn R= TRUE;

// NETWORK 8
GV.stHMI.stBatch_Ctrl.bCreate R= TRUE;
GV.stHMI.stBatch_Ctrl.bOpen R= TRUE;
GV.stHMI.stBatch_Ctrl.bCancel R= TRUE;
GV.stHMI.stBatch_Ctrl.bLoad R= TRUE;
GV.stHMI.stBatch_Ctrl.bLoadSP R= TRUE;
GV.stHMI.stBatch_Ctrl.bClose R= TRUE;

// NETWORK 9
GV.stHMI.stProcess_Ctrl.bLid_Open R= TRUE;
GV.stHMI.stProcess_Ctrl.bLid_Close R= TRUE;
GV.stHMI.stProcess_Ctrl.bOutlet_Open R= TRUE;
GV.stHMI.stProcess_Ctrl.bOutlet_Close R= TRUE;
GV.stHMI.stProcess_Ctrl.bSieve_SealOff R= TRUE;
GV.stHMI.stProcess_Ctrl.bSieve_SealOn R= TRUE;
GV.stHMI.stProcess_Ctrl.bTool_Raise R= TRUE;
GV.stHMI.stProcess_Ctrl.bTool_Lower R= TRUE;
GV.stHMI.stProcess_Ctrl.bMixer_FindPos R= TRUE;

// NETWORK 10
GV.stHMI.stMachine_Ctrl.bStart R= TRUE;
GV.stHMI.stMachine_Ctrl.bStop R= TRUE;
GV.stHMI.stMachine_Ctrl.bPause R= TRUE;

// NETWORK 11
GV.stHMI.stSP_Machine_Ctrl.bStart R= TRUE;
GV.stHMI.stSP_Machine_Ctrl.bStop R= TRUE;
GV.stHMI.stSP_Machine_Ctrl.bPause R= TRUE;

// NETWORK 12
GV.stHMI.stMachine_Ctrl.bNext R= TRUE;
GV.stHMI.stMachine_Ctrl.bPrevious R= TRUE;

// NETWORK 13
GV.stHMI.stProcess_Ctrl.bPump_Start R= TRUE;
GV.stHMI.stProcess_Ctrl.bPump_Stop R= TRUE;
GV.stHMI.stProcess_Ctrl.bMixer_Start R= TRUE;
GV.stHMI.stProcess_Ctrl.bMixer_Stop R= TRUE;
GV.stHMI.stProcess_Ctrl.bSieve_Start R= TRUE;
GV.stHMI.stProcess_Ctrl.bSieve_Stop R= TRUE;

// NETWORK 14
GV.stHMI.stProcess_Ctrl.bSP_Heater_Toggle R= TRUE;
GV.stHMI.stProcess_Ctrl.bSP_Mixer_Toggle R= TRUE;

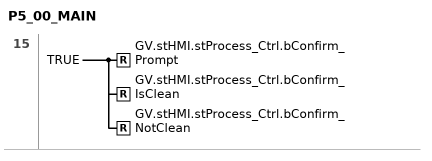
// NETWORK 15
GV.stHMI.stProcess_Ctrl.bConfirm_Prompt R= TRUE;
GV.stHMI.stProcess_Ctrl.bConfirm_IsClean R= TRUE;
GV.stHMI.stProcess_Ctrl.bConfirm_NotClean R= TRUE;

END_PROGRAM

// ---- POUs/5. HMI/P5_01_EnableControls.TcPOU
PROGRAM P5_01_EnableControls
VAR
	tonDisableNext			:TON;
	tonDisablePrev			:TON;
	tonDelayLid				:TON;
END_VAR
VAR // added by the converter: edge detectors and wires of the graphical bodies
    _w1 : BOOL;
END_VAR

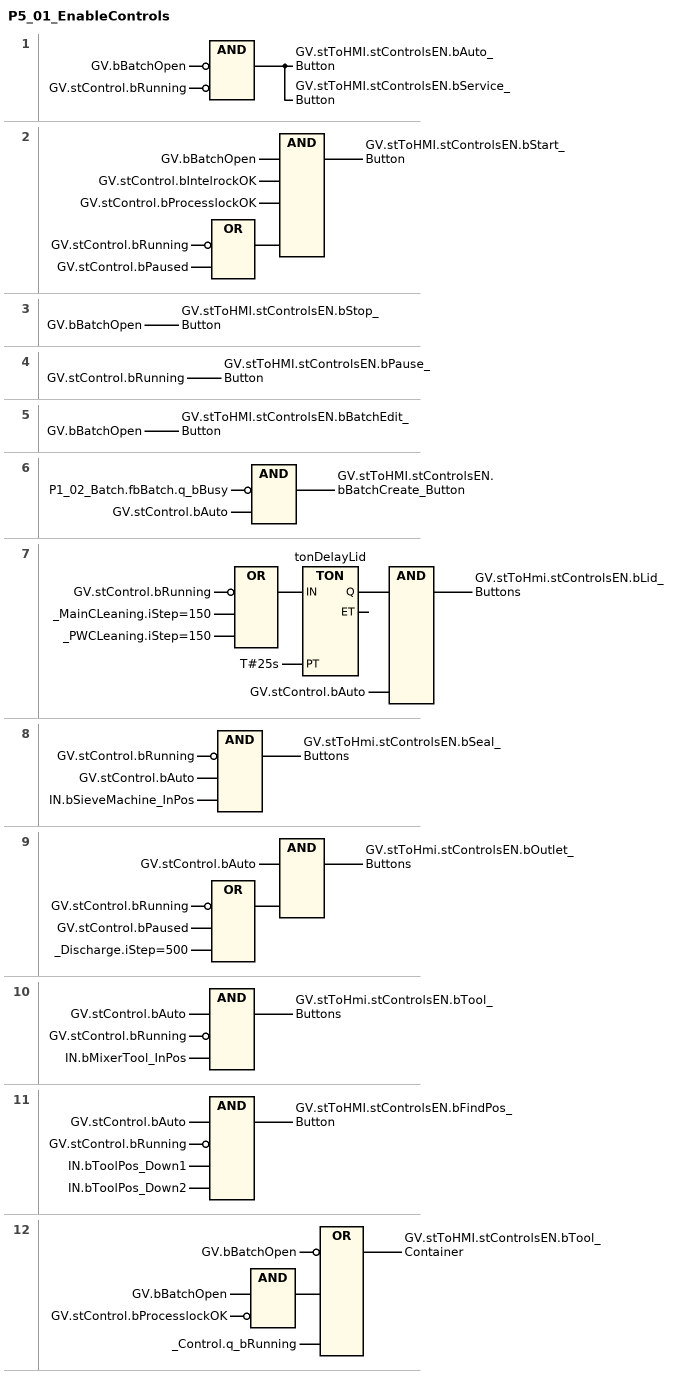
// NETWORK 1
_w1 := NOT GV.bBatchOpen AND NOT GV.stControl.bRunning;
GV.stToHMI.stControlsEN.bAuto_Button := _w1;
GV.stToHMI.stControlsEN.bService_Button := _w1;

// NETWORK 2
GV.stToHMI.stControlsEN.bStart_Button := GV.bBatchOpen AND GV.stControl.bIntelrockOK AND GV.stControl.bProcesslockOK AND (NOT GV.stControl.bRunning OR GV.stControl.bPaused);

// NETWORK 3
GV.stToHMI.stControlsEN.bStop_Button := GV.bBatchOpen;

// NETWORK 4
GV.stToHMI.stControlsEN.bPause_Button := GV.stControl.bRunning;

// NETWORK 5
GV.stToHMI.stControlsEN.bBatchEdit_Button := GV.bBatchOpen;

// NETWORK 6
GV.stToHMI.stControlsEN.bBatchCreate_Button := NOT P1_02_Batch.fbBatch.q_bBusy AND GV.stControl.bAuto;

// NETWORK 7
tonDelayLid(IN := NOT GV.stControl.bRunning OR (_MainCLeaning.iStep=150) OR (_PWCLeaning.iStep=150), PT := T#25s); // TON
GV.stToHmi.stControlsEN.bLid_Buttons := tonDelayLid.Q AND GV.stControl.bAuto;

// NETWORK 8
GV.stToHmi.stControlsEN.bSeal_Buttons := NOT GV.stControl.bRunning AND GV.stControl.bAuto AND IN.bSieveMachine_InPos;

// NETWORK 9
GV.stToHmi.stControlsEN.bOutlet_Buttons := GV.stControl.bAuto AND (NOT GV.stControl.bRunning OR GV.stControl.bPaused OR (_Discharge.iStep=500));

// NETWORK 10
GV.stToHmi.stControlsEN.bTool_Buttons := GV.stControl.bAuto AND NOT GV.stControl.bRunning AND IN.bMixerTool_InPos;

// NETWORK 11
GV.stToHMI.stControlsEN.bFindPos_Button := GV.stControl.bAuto AND NOT GV.stControl.bRunning AND IN.bToolPos_Down1 AND IN.bToolPos_Down2;

// NETWORK 12
GV.stToHMI.stControlsEN.bTool_Container := NOT GV.bBatchOpen OR GV.bBatchOpen AND NOT GV.stControl.bProcesslockOK OR _Control.q_bRunning;

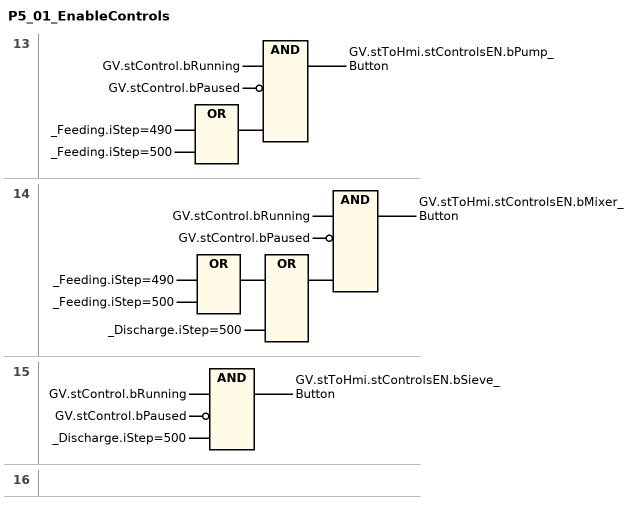
// NETWORK 13
GV.stToHmi.stControlsEN.bPump_Button := GV.stControl.bRunning AND NOT GV.stControl.bPaused AND ((_Feeding.iStep=490) OR (_Feeding.iStep=500));

// NETWORK 14
GV.stToHmi.stControlsEN.bMixer_Button := GV.stControl.bRunning AND NOT GV.stControl.bPaused AND (((_Feeding.iStep=490) OR (_Feeding.iStep=500)) OR (_Discharge.iStep=500));

// NETWORK 15
GV.stToHmi.stControlsEN.bSieve_Button := GV.stControl.bRunning AND NOT GV.stControl.bPaused AND (_Discharge.iStep=500);

// NETWORK 16

END_PROGRAM

// ---- POUs/5. HMI/P5_02_DiagramVisualisation.TcPOU
PROGRAM P5_02_DiagramVisualisation
VAR
END_VAR
VAR // added by the converter: edge detectors and wires of the graphical bodies
    _w1, _w2, _w3 : BOOL;
    _w4 : INT;
END_VAR

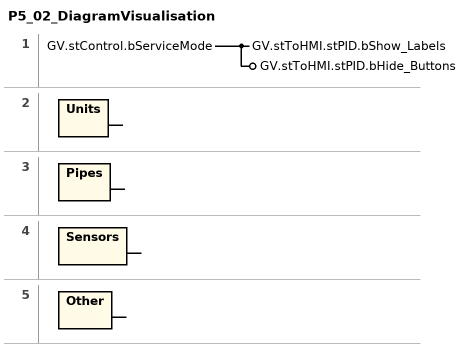
// NETWORK 1
_w1 := GV.stControl.bServiceMode;
GV.stToHMI.stPID.bShow_Labels := _w1;
GV.stToHMI.stPID.bHide_Buttons := NOT _w1;

// NETWORK 2
Units();

// NETWORK 3
Pipes();

// NETWORK 4
Sensors();

// NETWORK 5
Other();

ACTION Other:
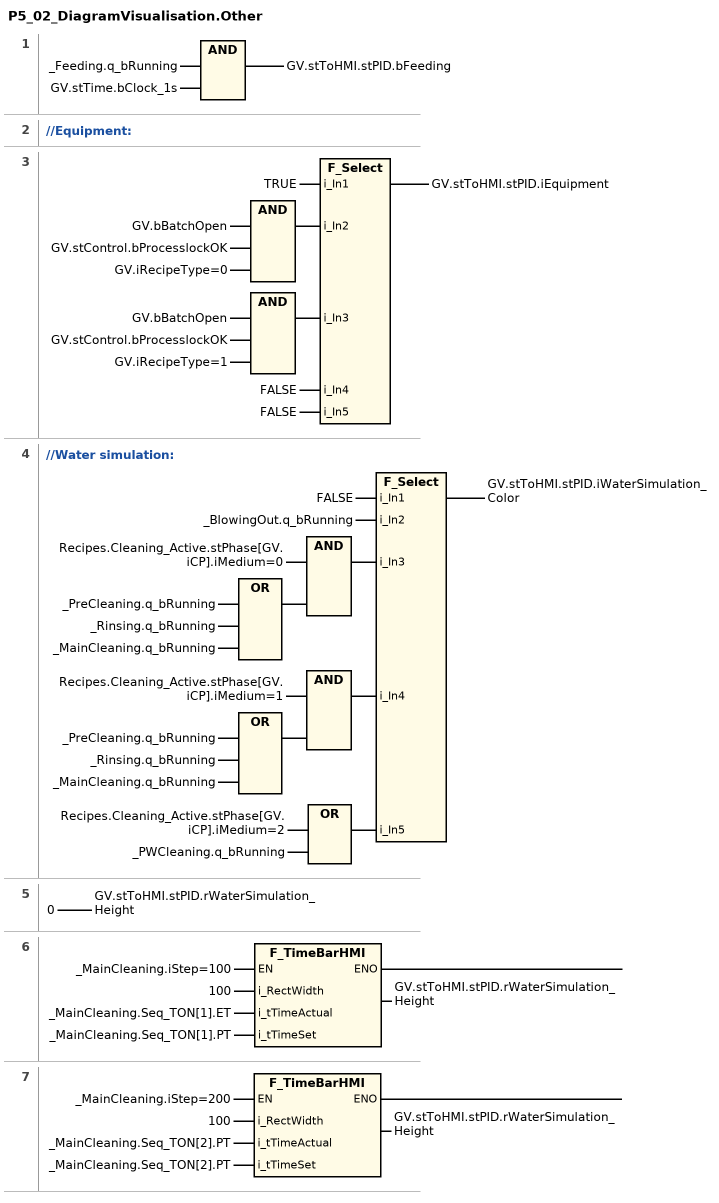
// NETWORK 1
GV.stToHMI.stPID.bFeeding := _Feeding.q_bRunning AND GV.stTime.bClock_1s;

// NETWORK 2
// label: //Equipment

// NETWORK 3
GV.stToHMI.stPID.iEquipment := F_Select(i_In1 := TRUE, i_In2 := GV.bBatchOpen AND GV.stControl.bProcesslockOK AND (GV.iRecipeType=0), i_In3 := GV.bBatchOpen AND GV.stControl.bProcesslockOK AND (GV.iRecipeType=1), i_In4 := FALSE, i_In5 := FALSE);

// NETWORK 4
// label: //Water simulation
GV.stToHMI.stPID.iWaterSimulation_Color := F_Select(i_In1 := FALSE, i_In2 := _BlowingOut.q_bRunning, i_In3 := (Recipes.Cleaning_Active.stPhase[GV.iCP].iMedium=0) AND (_PreCleaning.q_bRunning OR _Rinsing.q_bRunning OR _MainCleaning.q_bRunning), i_In4 := (Recipes.Cleaning_Active.stPhase[GV.iCP].iMedium=1) AND (_PreCleaning.q_bRunning OR _Rinsing.q_bRunning OR _MainCleaning.q_bRunning), i_In5 := (Recipes.Cleaning_Active.stPhase[GV.iCP].iMedium=2) OR _PWCleaning.q_bRunning);

// NETWORK 5
GV.stToHMI.stPID.rWaterSimulation_Height := 0;

// NETWORK 6
IF _MainCleaning.iStep=100 THEN
    GV.stToHMI.stPID.rWaterSimulation_Height := F_TimeBarHMI(i_RectWidth := 100, i_tTimeActual := _MainCleaning.Seq_TON[1].ET, i_tTimeSet := _MainCleaning.Seq_TON[1].PT);
END_IF

// NETWORK 7
IF _MainCleaning.iStep=200 THEN
    GV.stToHMI.stPID.rWaterSimulation_Height := F_TimeBarHMI(i_RectWidth := 100, i_tTimeActual := _MainCleaning.Seq_TON[2].PT, i_tTimeSet := _MainCleaning.Seq_TON[2].PT);
END_IF

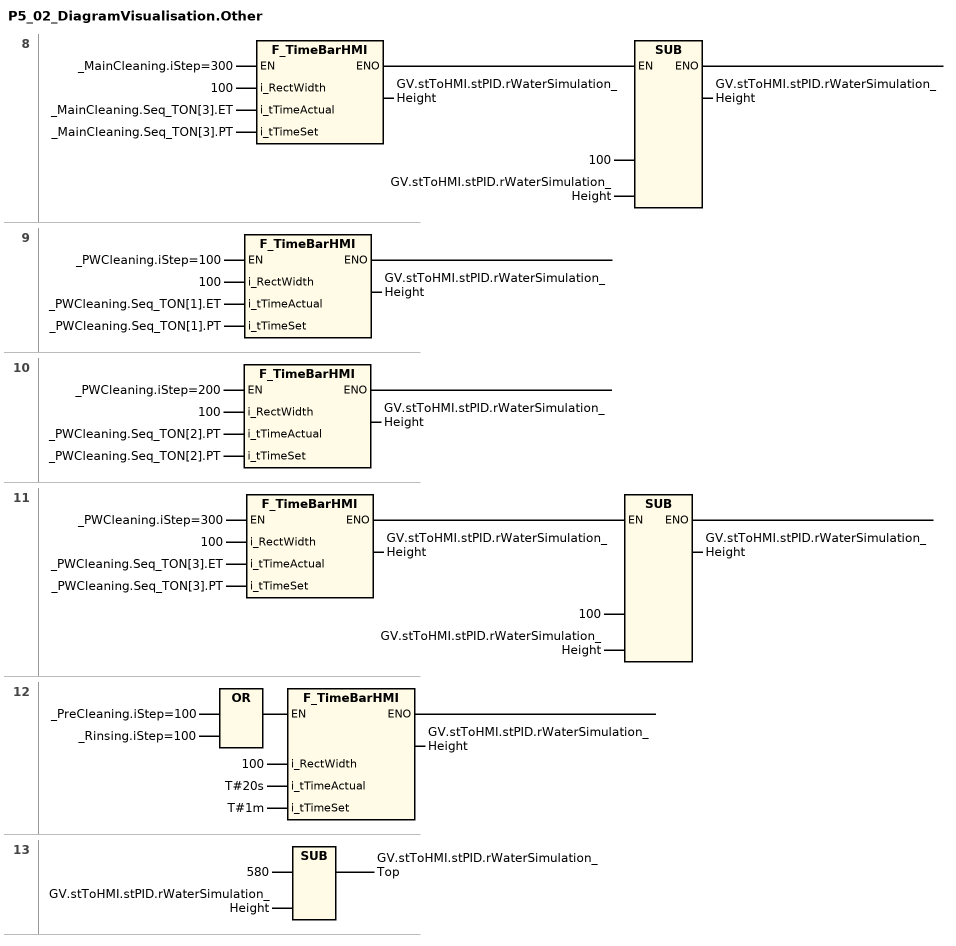
// NETWORK 8
_w2 := _MainCleaning.iStep=300;
IF _w2 THEN
    GV.stToHMI.stPID.rWaterSimulation_Height := F_TimeBarHMI(i_RectWidth := 100, i_tTimeActual := _MainCleaning.Seq_TON[3].ET, i_tTimeSet := _MainCleaning.Seq_TON[3].PT);
END_IF
IF _w2 THEN GV.stToHMI.stPID.rWaterSimulation_Height := 100 - GV.stToHMI.stPID.rWaterSimulation_Height; END_IF

// NETWORK 9
IF _PWCleaning.iStep=100 THEN
    GV.stToHMI.stPID.rWaterSimulation_Height := F_TimeBarHMI(i_RectWidth := 100, i_tTimeActual := _PWCleaning.Seq_TON[1].ET, i_tTimeSet := _PWCleaning.Seq_TON[1].PT);
END_IF

// NETWORK 10
IF _PWCleaning.iStep=200 THEN
    GV.stToHMI.stPID.rWaterSimulation_Height := F_TimeBarHMI(i_RectWidth := 100, i_tTimeActual := _PWCleaning.Seq_TON[2].PT, i_tTimeSet := _PWCleaning.Seq_TON[2].PT);
END_IF

// NETWORK 11
_w3 := _PWCleaning.iStep=300;
IF _w3 THEN
    GV.stToHMI.stPID.rWaterSimulation_Height := F_TimeBarHMI(i_RectWidth := 100, i_tTimeActual := _PWCleaning.Seq_TON[3].ET, i_tTimeSet := _PWCleaning.Seq_TON[3].PT);
END_IF
IF _w3 THEN GV.stToHMI.stPID.rWaterSimulation_Height := 100 - GV.stToHMI.stPID.rWaterSimulation_Height; END_IF

// NETWORK 12
IF (_PreCleaning.iStep=100) OR (_Rinsing.iStep=100) THEN
    GV.stToHMI.stPID.rWaterSimulation_Height := F_TimeBarHMI(i_RectWidth := 100, i_tTimeActual := T#20s, i_tTimeSet := T#1m);
END_IF

// NETWORK 13
GV.stToHMI.stPID.rWaterSimulation_Top := 580 - GV.stToHMI.stPID.rWaterSimulation_Height;
END_ACTION

ACTION Pipes:
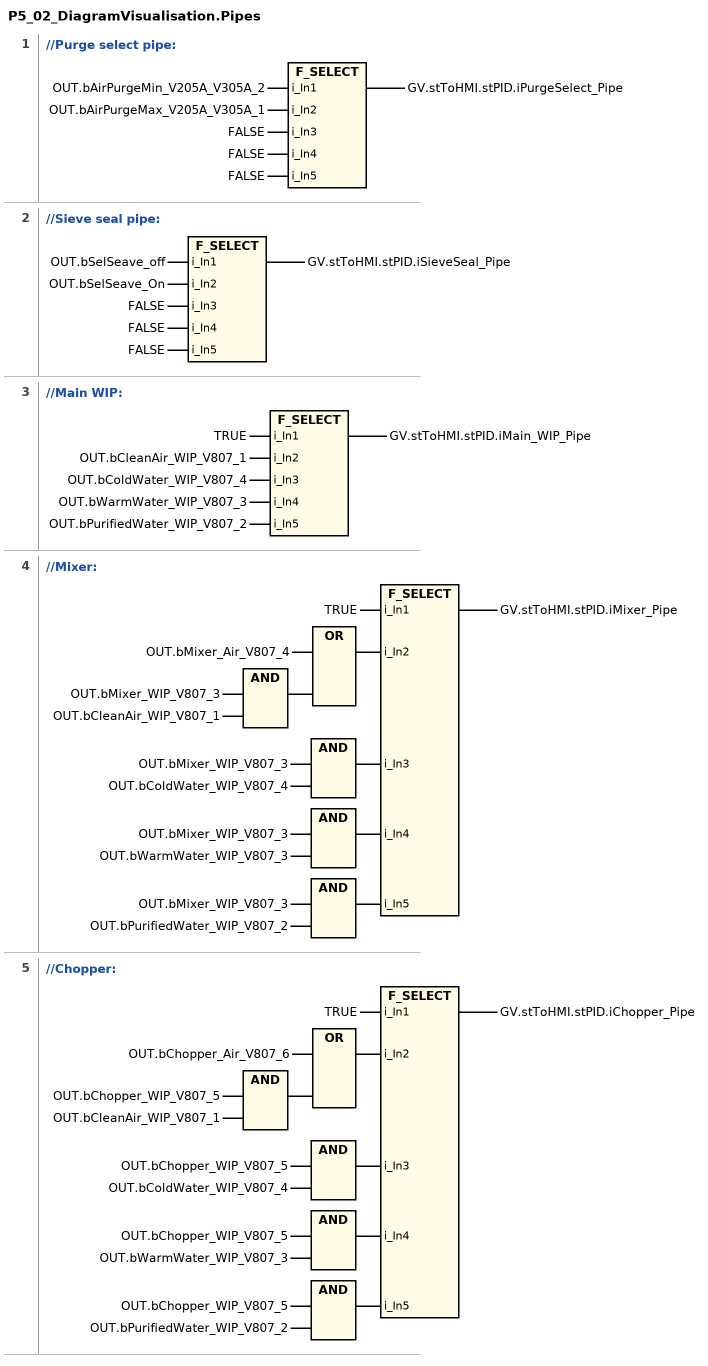
// NETWORK 1
// label: //Purge select pipe
GV.stToHMI.stPID.iPurgeSelect_Pipe := F_SELECT(i_In1 := OUT.bAirPurgeMin_V205A_V305A_2, i_In2 := OUT.bAirPurgeMax_V205A_V305A_1, i_In3 := FALSE, i_In4 := FALSE, i_In5 := FALSE);

// NETWORK 2
// label: //Sieve seal pipe
GV.stToHMI.stPID.iSieveSeal_Pipe := F_SELECT(i_In1 := OUT.bSelSeave_off, i_In2 := OUT.bSelSeave_On, i_In3 := FALSE, i_In4 := FALSE, i_In5 := FALSE);

// NETWORK 3
// label: //Main WIP
GV.stToHMI.stPID.iMain_WIP_Pipe := F_SELECT(i_In1 := TRUE, i_In2 := OUT.bCleanAir_WIP_V807_1, i_In3 := OUT.bColdWater_WIP_V807_4, i_In4 := OUT.bWarmWater_WIP_V807_3, i_In5 := OUT.bPurifiedWater_WIP_V807_2);

// NETWORK 4
// label: //Mixer
GV.stToHMI.stPID.iMixer_Pipe := F_SELECT(i_In1 := TRUE, i_In2 := OUT.bMixer_Air_V807_4 OR OUT.bMixer_WIP_V807_3 AND OUT.bCleanAir_WIP_V807_1, i_In3 := OUT.bMixer_WIP_V807_3 AND OUT.bColdWater_WIP_V807_4, i_In4 := OUT.bMixer_WIP_V807_3 AND OUT.bWarmWater_WIP_V807_3, i_In5 := OUT.bMixer_WIP_V807_3 AND OUT.bPurifiedWater_WIP_V807_2);

// NETWORK 5
// label: //Chopper
GV.stToHMI.stPID.iChopper_Pipe := F_SELECT(i_In1 := TRUE, i_In2 := OUT.bChopper_Air_V807_6 OR OUT.bChopper_WIP_V807_5 AND OUT.bCleanAir_WIP_V807_1, i_In3 := OUT.bChopper_WIP_V807_5 AND OUT.bColdWater_WIP_V807_4, i_In4 := OUT.bChopper_WIP_V807_5 AND OUT.bWarmWater_WIP_V807_3, i_In5 := OUT.bChopper_WIP_V807_5 AND OUT.bPurifiedWater_WIP_V807_2);

